FUNCTION_BLOCK FB_EcatDiag
VAR_INPUT
	i_AMSNetId	:	AMSNETID; //Connect this to an AMSNETID structure as a PLC input. Then link the input to the AMSNETID name in the master info.
	i_xFirstPass	:	BOOL;
END_VAR
VAR_OUTPUT
	q_xAllStatesGood	:	BOOL;
END_VAR
VAR
	sNetId : T_AmsNetId;
	astTermStates : ARRAY[1..256] OF ST_EcSlaveState;
	
	fbGetAllSlaveStates     : FB_EcGetAllSlaveStates;
	ftReset	: F_TRIG;
	
	iterator: INT;
END_VAR

//Create the net ID string
sNetID := F_CreateAmsNetId(i_AMSNetId);

//Query the state of all terminals, collect in astTermStates
ftReset(CLK:=fbGetAllSlaveStates.bBusy OR i_xFirstPass);
fbGetAllSlaveStates.bExecute := ftReset.Q;
fbGetAllSlaveStates(sNetId:=sNetId, pStateBuf := ADR(astTermStates), cbBufLen:=SIZEOF(astTermStates));
//Keep checking...

//Cycle through each entry in the array and check if we have anyone not in OP and that the link state is good.
// If so, then set our global IO bad boolean.
IF fbGetAllSlaveStates.nSlaves > 0 THEN
	q_xAllStatesGood := TRUE;
FOR iterator := 1 TO (fbGetAllSlaveStates.nSlaves -1) BY 1
	DO
	IF NOT( (astTermStates[iterator].deviceState = EC_DEVICE_STATE_OP) AND (astTermStates[iterator].linkState = EC_LINK_STATE_OK)) THEN
		q_xAllStatesGood := FALSE;
	END_IF
END_FOR
END_IF

END_FUNCTION_BLOCK

(* stored: Version 1.1.0.1, ProductVersion 3.1.0.26
   POU FB_EcatDiag: Id {5f761df3-17d1-44c1-84cd-865068aed9a8} *)
